GLOBALCONSTANTS DefaultPool_Horse (* Global constants *)
  PACKAGE Uebungen::const::UT::Horse;
  VAR_GLOBAL CONSTANT
    ISO_DESIGNATOR_WIDTH : UINT := 80;
    ISO_DESIGNATOR_HEIGHT : UINT := 80;
    ISO_MASK_SIZE : UINT := 480;
    ISO_VERSION_LABEL : STRING;
    MASK_WIDTH : UINT := 480;
    MASK_HEIGHT : UINT := 480;
    WorkingSet : UINT := 0;
    DataMask_Main : UINT := 1000;
    DataMask_invisible : UINT := 1001;
    frame_00 : UINT := 20000;
    frame_01 : UINT := 20001;
    frame_02 : UINT := 20002;
    frame_03 : UINT := 20003;
    frame_04 : UINT := 20004;
    frame_05 : UINT := 20005;
    frame_06 : UINT := 20006;
    frame_07 : UINT := 20007;
    frame_08 : UINT := 20008;
    frame_09 : UINT := 20009;
    frame_10 : UINT := 20010;
    frame_11 : UINT := 20011;
    frame_12 : UINT := 20012;
    frame_13 : UINT := 20013;
    frame_14 : UINT := 20014;
    frame_15 : UINT := 20015;
    frame_16 : UINT := 20016;
    frame_17 : UINT := 20017;
    frame_18 : UINT := 20018;
    frame_19 : UINT := 20019;
    frame_20 : UINT := 20020;
    frame_21 : UINT := 20021;
    frame_22 : UINT := 20022;
    frame_23 : UINT := 20023;
    frame_24 : UINT := 20024;
    frame_25 : UINT := 20025;
    frame_26 : UINT := 20026;
    frame_27 : UINT := 20027;
    frame_28 : UINT := 20028;
    frame_29 : UINT := 20029;
    frame_30 : UINT := 20030;
    frame_31 : UINT := 20031;
    ws_pic : UINT := 20532;
    ObjectPointer_Horse : UINT := 27000;
  END_VAR
END_GLOBALCONSTANTS
